(* IEC 61131-3 sources: plc-vscode/tests/st/test-ready/trust-platform/examples/filling_line/src, 7 files *)

(* ---- Types.st ---- *)
TYPE
    LevelMode : (Stopped, Filling, Draining);
END_TYPE

(* ---- Interfaces.st ---- *)
INTERFACE IValve
    METHOD Open : BOOL
    END_METHOD

    METHOD Close : BOOL
    END_METHOD

    PROPERTY IsOpen : BOOL
        GET
        END_GET
    END_PROPERTY
END_INTERFACE

INTERFACE IPump
    METHOD Start : BOOL
    END_METHOD

    METHOD Stop : BOOL
    END_METHOD

    PROPERTY IsRunning : BOOL
        GET
        END_GET
    END_PROPERTY

    PROPERTY Speed : INT
        GET
        END_GET
        SET
        END_SET
    END_PROPERTY
END_INTERFACE

(* ---- LevelController.st ---- *)
FUNCTION_BLOCK LevelController
VAR_INPUT
    LevelPct : REAL;
    StartCmd : BOOL;
    StopCmd : BOOL;
END_VAR
VAR_OUTPUT
    FillCmd : BOOL;
    DrainCmd : BOOL;
    Mode : LevelMode;
END_VAR
VAR
    Target : REAL := 70.0;
    Hysteresis : REAL := 5.0;
END_VAR

IF StopCmd THEN
    Mode := LevelMode#Stopped;
ELSIF StartCmd THEN
    IF LevelPct < Target - Hysteresis THEN
        Mode := LevelMode#Filling;
    ELSIF LevelPct > Target + Hysteresis THEN
        Mode := LevelMode#Draining;
    ELSE
        Mode := LevelMode#Stopped;
    END_IF;
END_IF;

FillCmd := Mode = LevelMode#Filling;
DrainCmd := Mode = LevelMode#Draining;
END_FUNCTION_BLOCK

(* ---- PumpDrive.st ---- *)
FUNCTION_BLOCK PumpDrive IMPLEMENTS IPump
VAR
    RunningValue : BOOL;
    SpeedValue : INT;
END_VAR

METHOD PUBLIC Start : BOOL
    RunningValue := TRUE;
    Start := RunningValue;
END_METHOD

METHOD PUBLIC Stop : BOOL
    RunningValue := FALSE;
    Stop := RunningValue;
END_METHOD

PUBLIC PROPERTY IsRunning : BOOL
    GET
        IsRunning := RunningValue;
    END_GET
    SET
    END_SET
END_PROPERTY

PUBLIC PROPERTY Speed : INT
    GET
        Speed := SpeedValue;
    END_GET
    SET
        SpeedValue := Speed;
    END_SET
END_PROPERTY
END_FUNCTION_BLOCK

(* ---- ValveActuator.st ---- *)
FUNCTION_BLOCK ValveActuator IMPLEMENTS IValve
VAR
    OpenState : BOOL;
END_VAR

METHOD PUBLIC Open : BOOL
    OpenState := TRUE;
    Open := OpenState;
END_METHOD

METHOD PUBLIC Close : BOOL
    OpenState := FALSE;
    Close := OpenState;
END_METHOD

PUBLIC PROPERTY IsOpen : BOOL
    GET
        IsOpen := OpenState;
    END_GET
END_PROPERTY
END_FUNCTION_BLOCK

(* ---- Configuration.st ---- *)
CONFIGURATION FillingLine
TASK Cycle (INTERVAL := T#50ms, PRIORITY := 1);
PROGRAM P1 WITH Cycle : MainProgram;
VAR_CONFIG
    P1.StartCmd AT %IX0.0 : BOOL;
    P1.StopCmd AT %IX0.1 : BOOL;
    P1.LevelRaw AT %IW0 : INT;
    P1.FillValveOut AT %QX0.0 : BOOL;
    P1.DrainValveOut AT %QX0.1 : BOOL;
    P1.PumpSpeedOut AT %QW0 : INT;
END_VAR
END_CONFIGURATION

(* ---- Main.st ---- *)
PROGRAM MainProgram
VAR
    StartCmd : BOOL;
    StopCmd : BOOL;
    LevelRaw : INT;
    FillValveOut : BOOL;
    DrainValveOut : BOOL;
    PumpSpeedOut : INT;

    LevelPct : REAL;
    Ctrl : LevelController;
END_VAR

LevelPct := INT_TO_REAL(LevelRaw) * 0.1;

Ctrl(LevelPct := LevelPct, StartCmd := StartCmd, StopCmd := StopCmd);

IF Ctrl.FillCmd THEN
    FillValveOut := TRUE;
    DrainValveOut := FALSE;
    PumpSpeedOut := INT#800;
ELSIF Ctrl.DrainCmd THEN
    FillValveOut := FALSE;
    DrainValveOut := TRUE;
    PumpSpeedOut := INT#600;
ELSE
    FillValveOut := FALSE;
    DrainValveOut := FALSE;
    PumpSpeedOut := INT#0;
END_IF;
END_PROGRAM
